PROGRAM PLC_PRG
VAR
	//Visualisation 	
	mxButtonPaus	: BOOL;

	mxAuto			: BOOL;

	//Internal use
	mxStart: BOOL;
	mxDone: BOOL;
	
	//Motion Function Blocks
	fbGantryStatus: GantryStatus;

	fbGantryPick_1: GantryPick;
	fbGantryLeave_2: GantryLeave;

	nPickStation: INT := 1;
	nPickPosition: INT := 1;
	nLeaveStation: INT := 1;
	nLeavePosition: INT := 2;
END_VAR
VAR // added by the converter: edge detectors and wires of the graphical bodies
    _w1, _w2 : BOOL;
END_VAR

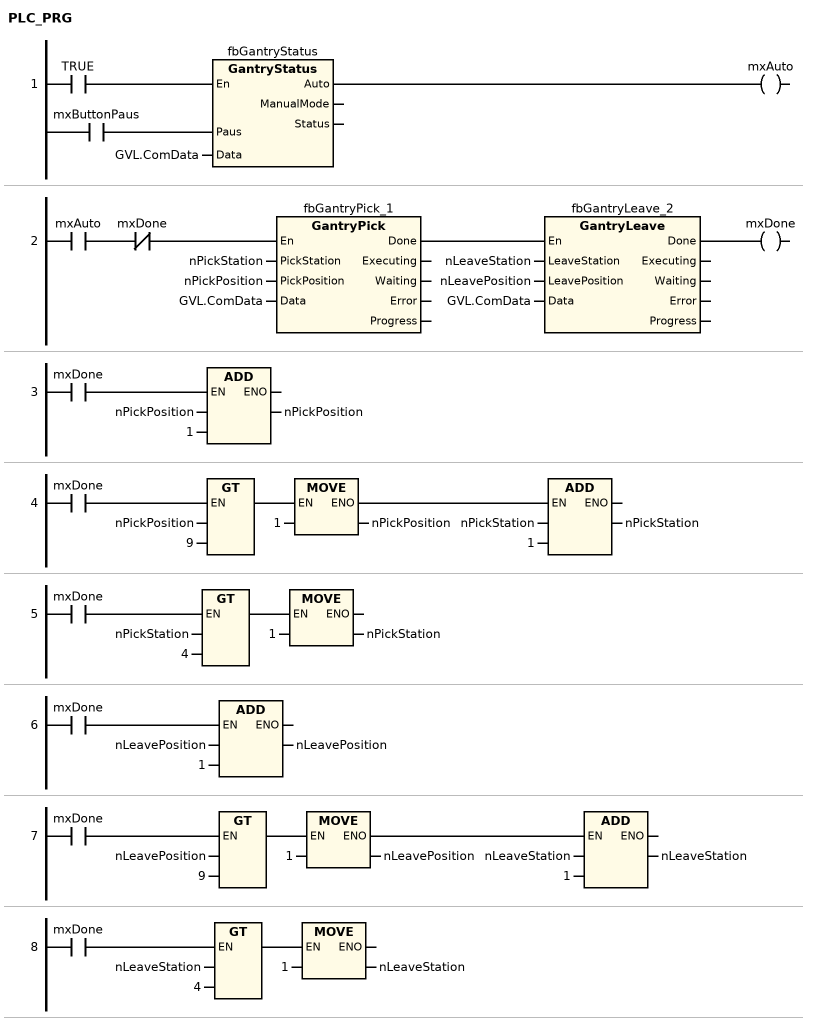
// NETWORK 1
fbGantryStatus(En := TRUE, Paus := mxButtonPaus, Data := GVL.ComData); // GantryStatus
mxAuto := fbGantryStatus.Auto;

// NETWORK 2
fbGantryPick_1(
    En := mxAuto AND NOT mxDone,
    PickStation := nPickStation,
    PickPosition := nPickPosition,
    Data := GVL.ComData); // GantryPick
fbGantryLeave_2(
    En := fbGantryPick_1.Done,
    LeaveStation := nLeaveStation,
    LeavePosition := nLeavePosition,
    Data := GVL.ComData); // GantryLeave
mxDone := fbGantryLeave_2.Done;

// NETWORK 3
IF mxDone THEN nPickPosition := nPickPosition + 1; END_IF

// NETWORK 4
_w1 := mxDone AND nPickPosition > 9;
IF _w1 THEN nPickPosition := 1; END_IF
IF _w1 THEN nPickStation := nPickStation + 1; END_IF

// NETWORK 5
IF mxDone AND nPickStation > 4 THEN nPickStation := 1; END_IF

// NETWORK 6
IF mxDone THEN nLeavePosition := nLeavePosition + 1; END_IF

// NETWORK 7
_w2 := mxDone AND nLeavePosition > 9;
IF _w2 THEN nLeavePosition := 1; END_IF
IF _w2 THEN nLeaveStation := nLeaveStation + 1; END_IF

// NETWORK 8
IF mxDone AND nLeaveStation > 4 THEN nLeaveStation := 1; END_IF

END_PROGRAM

(* stored: Version 1.1.0.1, ProductVersion 3.1.4022.12
   POU PLC_PRG: Id {04ec82fb-e5b1-40a1-85a5-368d0068671a}, SpecialFunc None *)
